FUNCTION_BLOCK PUBLIC ABSTRACT FB_ManualUiBase IMPLEMENTS I_ManualUi
VAR_INPUT
	// object name
	stName 					: ST_Text;
	// objekts index
	diObjectIndex			: DINT;
	// selected object index in hmi 
	diSelectedObjectIndex	: DINT;
	/// manual mode enable
	bEnableManual			: BOOL;
	/// device BMK
	stBmk					: ST_Text;
	// state object
	stStateObject			: REFERENCE TO ST_Object_Item;
END_VAR
VAR_OUTPUT
	/// Fehler
	bError				: BOOL;
	/// Fehlertext
	stErrorText			: ST_Text;
	/// Warnung
	bWarning			: BOOL;
	/// Warnungstext
	stWarnText			: ST_Text;
END_VAR
VAR
	bManualActive			: BOOL;
END_VAR

// to be subclassed..

METHOD M_SetStateObject : BOOL
VAR_IN_OUT
	stStateObjectRef	: ST_Object_Item;
END_VAR
stStateObject REF= stStateObjectRef;
END_METHOD

PROPERTY Name : ST_Text
GET
Name := stName;
END_GET
END_PROPERTY

PROPERTY ObjectIndex : DINT
GET
ObjectIndex := diObjectIndex;
END_GET
SET
diObjectIndex := ObjectIndex;
END_SET
END_PROPERTY

END_FUNCTION_BLOCK

(* stored: Version 1.1.0.1
   POU FB_ManualUiBase: Id {196208e1-dc9f-43f2-b660-5fb08a661390}, SpecialFunc None
   Method M_SetStateObject: Id {01d1373c-6efa-494d-985c-1dd29976e8b4}
   Property Name: Id {2dfd67b3-41ac-4b63-b2fd-91d143adbd57}
   Get Get: Id {62876ca2-1ff8-4df3-b2f0-0f80e29201c6}
   Property ObjectIndex: Id {4c3b081c-5064-4006-8595-2088de9cdb54}
   Get Get: Id {d1aafeca-6dd0-41e1-b08c-71e218181210}
   Set Set: Id {c17f20d2-7a5e-4c33-aaa7-befb6becf2b1} *)
